FUNCTION_BLOCK ShelfElement IMPLEMENTS IShelfElement
VAR_INPUT
END_VAR
VAR_OUTPUT
END_VAR
VAR
	_id: STRING(ID_SIZE);
	_isOccupied: BOOL := FALSE;
END_VAR
VAR CONSTANT
	ID_SIZE: INT := 23;
END_VAR

PROPERTY id : STRING(ID_SIZE)
GET
id := THIS^._id;
END_GET
SET
THIS^._id := id;
END_SET
END_PROPERTY

{warning 'Add property implementation'}
PROPERTY isOccupied : BOOL
GET
isOccupied := THIS^._isOccupied;
END_GET
SET
THIS^._isOccupied := isOccupied;
END_SET
END_PROPERTY

END_FUNCTION_BLOCK

(* stored: Version 1.1.0.1
   POU ShelfElement: Id {6f2a0f5e-9c15-4f74-a25b-4b294e8cf477}, SpecialFunc None
   Property id: Id {c916ffda-12ce-4694-bf43-76f1f3687346}
   Get Get: Id {2cdcb989-e356-4d18-8c1d-d89233812b74}
   Set Set: Id {f10b9992-36e4-4a98-8494-a84393832637}
   Property isOccupied: Id {2a504b2a-6c12-4377-b320-e920663caff7}
   Get Get: Id {a589052c-4414-45b6-9adf-592b846cccd7}
   Set Set: Id {061a3683-f41d-4aa8-b9fc-8f65e2212c33} *)
